FUNCTION_BLOCK FB_Drive
VAR_IN_OUT
	bInHome: BOOL;
END_VAR
VAR_INPUT
	/// component active flag
	bActive: BOOL;
	/// Objekt Name (BMK)
	stName				:ST_Text;
	/// Sicherheit = Freigabe von Bewegungen
	bSafetyOk			:BOOL;
	/// Motorschutz OK
	bMotorprotectionOk		:BOOL;

	// Hand
	///Objekt Index
	diObjectIndex: DINT;
	///Ausgewähltes Objekt in der Visu
	diSelectedObjectIndex	:DINT;
	/// Gibt den Handbetrieb frei
	bEnableManual: BOOL;
	// Handbetrieb nach GRST
	bManual_Reverse: BOOL;
	/// Handbetrieb nach AST
	bManual_Forward: BOOL;
	///	 Handbetrieb Stop
	bManual_Stop :BOOL;
	//	Type Handbetrieb
	// 1 = Tippen
	// 2 = Speichern
	iType : INT;
	
	///	Zus. Freigabe für HP Ausgang schalten	
	bFreigabe_Reverse: BOOL := TRUE;
	///	Zus. Freigabe für WP Ausgang schalten	
	bFreigabe_Forward: BOOL := TRUE;
END_VAR
VAR_OUTPUT	
	/// Summenfehler
	bError		:BOOL;
	/// Fehlerinformation
	sErrText	:ST_Text;
	/// 0=Undefiniert
	/// 1=Fehler
	/// 2=Stillstand OK
	/// 3=Vorwärts
	///	4=Rückwärts 
	iStatus: INT;	

	bInit_OK: BOOL;
	
	bDrive_Reverse_Out: BOOL;
	bDrive_Forward_Out: BOOL;
END_VAR
VAR
	iTypeOld : INT;
	tofForward: TOF;
	tofReverse: TOF;
	
	bDrive_Reverse: BOOL;
	bDrive_Forward: BOOL;
END_VAR

(*FB Drive für Antriebe*)
(*Erstellt von Stephan Schöchtner RMTH GmbH*)
(*21.März.2018*)

tofForward();
tofForward.IN := bManual_Forward;

tofReverse();
tofReverse.IN := bManual_Reverse;


// Initialisierung
IF NOT bInit_OK THEN
	M_Init();	
	bInit_OK :=TRUE;
END_IF

sERRText := CONST.stTextListGlobal.stText_notext;

//Fehler
bError := FALSE;
IF NOT bMotorprotectionOK THEN
	bError := TRUE;
	sErrText := F_CreateDynText("Motorschutz", 0);
END_IF

// Bei Typumschaltung im laufenden Betrieb STOP
IF iType <> iTypeOld THEN
	iTypeOld := iType;
	M_Stop();
END_IF

IF (diObjectIndex = diSelectedObjectIndex) THEN
	// Tippen mit Wendeschützumschaltung und Typumschaltung
	CASE iType OF	//Tippen
	
		1:
			IF bManual_Forward AND NOT bManual_Stop THEN
				bDrive_Reverse := FALSE;
				IF NOT tofReverse.Q THEN
					M_Start_Forward();
				END_IF
			ELSIF bManual_Reverse AND NOT bManual_Stop THEN
				bDrive_Forward := FALSE;
				IF NOT tofForward.Q THEN
					M_Start_Reverse();
				END_IF
			ELSE
				M_Stop();
				//M_Start_Forward := FALSE;
				//M_Start_Reverse := FALSE;
			END_IF
		2:						//Speichern
			IF bManual_Forward AND NOT bManual_Stop THEN
				bDrive_Reverse := FALSE;
				IF NOT tofReverse.Q THEN
					M_Start_Forward();
				END_IF
			ELSIF bManual_Reverse AND NOT bManual_Stop THEN
				bDrive_Forward := FALSE;
				IF NOT tofForward.Q THEN
					M_Start_Reverse();
				END_IF
			END_IF
			IF bManual_Stop THEN
				M_Stop();
				//M_Start_Forward := FALSE;
				//M_Start_Reverse := FALSE;
			END_IF	
	ELSE
		//no type selected
		bError := TRUE;
		sErrText := F_CreateDynText("Handbetriebstyp falsch", 0);
		M_Stop();
	END_CASE
END_IF

IF bError THEN
	istatus := 1;
ELSIF NOT bDrive_Forward AND NOT bDrive_Reverse THEN
	iStatus := 2;
ELSIF bDrive_Forward THEN
	iStatus := 3;
ELSIF bDrive_Reverse THEN
	iStatus := 4;
END_IF


bDrive_Reverse_Out:= bDrive_Reverse AND bFreigabe_Reverse AND bSafetyOk AND bMotorprotectionOk;
bDrive_Forward_Out:= bDrive_Forward AND bFreigabe_Forward AND bSafetyOk AND bMotorprotectionOk;

IF NOT bSafetyOk THEN
	bDrive_Reverse:=FALSE;
	bDrive_Reverse_Out:=FALSE;

	bDrive_Forward:=FALSE;
	bDrive_Forward_Out:=FALSE;	
END_IF


//Wegfahrsperre
IF bError THEN
	M_Stop();
END_IF

METHOD M_Init : BOOL
VAR_INPUT
END_VAR
bDrive_Forward := FALSE;
bDrive_Reverse := FALSE;
tofForward.IN := FALSE;
tofForward.PT := T#150MS;
tofReverse.IN := FALSE;
tofReverse.PT := T#150MS;
END_METHOD

METHOD M_Reset : BOOL
VAR_INPUT
END_VAR
END_METHOD

METHOD M_Start_Forward : BOOL
VAR_INPUT
END_VAR
bDrive_Reverse := FALSE;
bDrive_Forward := TRUE;
END_METHOD

METHOD M_Start_Reverse : BOOL
VAR_INPUT
END_VAR
bDrive_Reverse := TRUE;
bDrive_Forward := FALSE;
END_METHOD

METHOD M_Stop : BOOL
VAR_INPUT
END_VAR
	bDrive_Reverse := FALSE;
	bDrive_Forward := FALSE;
END_METHOD

END_FUNCTION_BLOCK

(* stored: Version 1.1.0.1, ProductVersion 3.1.4024.4
   POU FB_Drive: Id {b811c766-f891-4e79-8b19-fc9f1052191b}, SpecialFunc None
   Method M_Init: Id {f8a224e2-5caa-475f-b0f3-eea92b648e57}
   Method M_Reset: Id {00f9d4a6-42dd-4266-ba47-7d656b00a099}
   Method M_Start_Forward: Id {7681f5a2-71df-4d3f-962a-7a1e7dc0fd04}
   Method M_Start_Reverse: Id {ceb8f507-bede-4b18-8437-757cc93c7b40}
   Method M_Stop: Id {438855a6-7d63-40fe-b81f-77e7427f4a86} *)
